Staubli VAL3: Vakuumgreifer.dtx

frame StaubliTX240Base = {x=0.000, y=0.000, z=0.000, rx=-0.000, ry=0.000, rz=-0.000, fatherId=world[0]}
dio dVacuum = {link=98FE10BA-0446-4B8A-A8CF-35B98F42725A}
tool tCurrentTool = {x=0.000, y=0.000, z=78.000, rx=-0.000, ry=0.000, rz=-0.000, fatherId=flange[0], ioLink=98FE10BA-0446-4B8A-A8CF-35B98F42725A}
mdesc mCurrentSpeed
pointRx pPointRx1 = {}
pointRx pPointRx2 = {}
